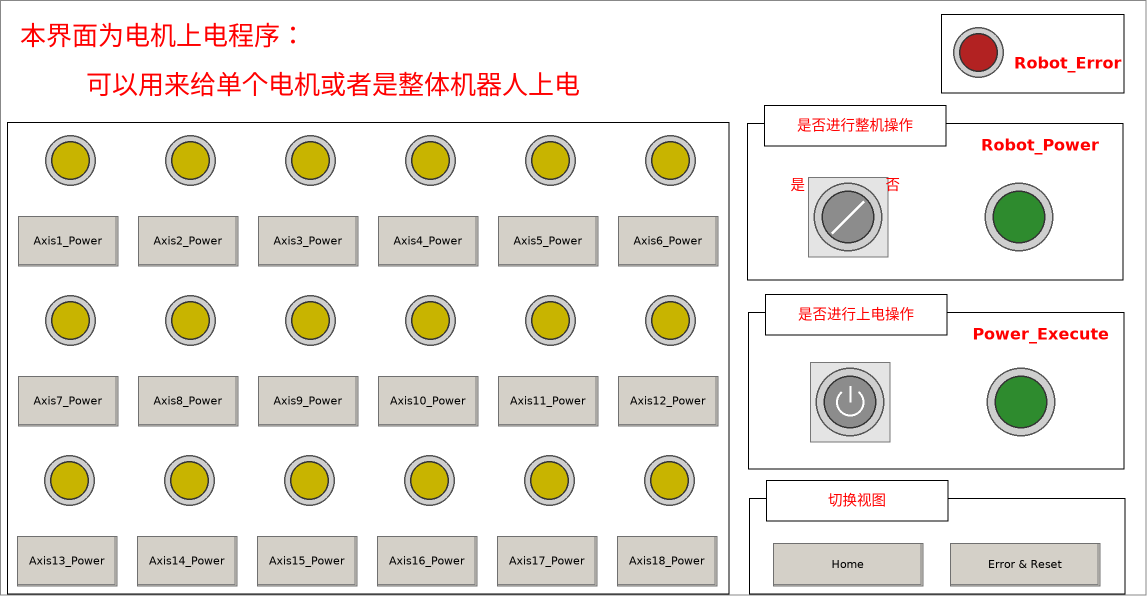
VISUALIZATION Visu_Power  // 1147x596
    Label (987,37 154x32), "Robot_Error"
    Rectangle (7,122 722x472)
    Lamp1 (40,131 61x59), variable: MAIN.Power_Status[1], style: Lamp-Lamp1-Yellow
    Lamp1 (160,131 61x59), variable: MAIN.Power_Status[2], style: Lamp-Lamp1-Yellow
    Lamp1 (280,131 61x59), variable: MAIN.Power_Status[3], style: Lamp-Lamp1-Yellow
    Lamp1 (400,131 61x59), variable: MAIN.Power_Status[4], style: Lamp-Lamp1-Yellow
    Lamp1 (520,131 61x59), variable: MAIN.Power_Status[5], style: Lamp-Lamp1-Yellow
    Lamp1 (640,131 61x59), variable: MAIN.Power_Status[6], style: Lamp-Lamp1-Yellow
    Button (18,216 100x50), "Axis1_Power"
        toggle MAIN.Axis_Power[1]
    Button (138,216 100x50), "Axis2_Power"
        toggle MAIN.Axis_Power[2]
    Button (258,216 100x50), "Axis3_Power"
        toggle MAIN.Axis_Power[3]
    Button (378,216 100x50), "Axis4_Power"
        toggle MAIN.Axis_Power[4]
    Button (498,216 100x50), "Axis5_Power"
        toggle MAIN.Axis_Power[5]
    Button (618,216 100x50), "Axis6_Power"
        toggle MAIN.Axis_Power[6]
    Lamp1 (40,291 61x59), variable: MAIN.Power_Status[7], style: Lamp-Lamp1-Yellow
    Lamp1 (160,291 61x59), variable: MAIN.Power_Status[8], style: Lamp-Lamp1-Yellow
    Lamp1 (280,291 61x59), variable: MAIN.Power_Status[9], style: Lamp-Lamp1-Yellow
    Lamp1 (400,291 61x59), variable: MAIN.Power_Status[10], style: Lamp-Lamp1-Yellow
    Lamp1 (520,291 61x59), variable: MAIN.Power_Status[11], style: Lamp-Lamp1-Yellow
    Lamp1 (640,291 61x59), variable: MAIN.Power_Status[12], style: Lamp-Lamp1-Yellow
    Button (18,376 100x50), "Axis7_Power"
        toggle MAIN.Axis_Power[7]
    Button (138,376 100x50), "Axis8_Power"
        toggle MAIN.Axis_Power[8]
    Button (258,376 100x50), "Axis9_Power"
        toggle MAIN.Axis_Power[9]
    Button (378,376 100x50), "Axis10_Power"
        toggle MAIN.Axis_Power[10]
    Button (498,376 100x50), "Axis11_Power"
        toggle MAIN.Axis_Power[11]
    Button (618,376 100x50), "Axis12_Power"
        toggle MAIN.Axis_Power[12]
    Lamp1 (39,451 61x59), variable: MAIN.Power_Status[13], style: Lamp-Lamp1-Yellow
    Lamp1 (159,451 61x59), variable: MAIN.Power_Status[14], style: Lamp-Lamp1-Yellow
    Lamp1 (279,451 61x59), variable: MAIN.Power_Status[15], style: Lamp-Lamp1-Yellow
    Lamp1 (399,451 61x59), variable: MAIN.Power_Status[16], style: Lamp-Lamp1-Yellow
    Lamp1 (519,451 61x59), variable: MAIN.Power_Status[17], style: Lamp-Lamp1-Yellow
    Lamp1 (639,451 61x59), variable: MAIN.Power_Status[18], style: Lamp-Lamp1-Yellow
    Button (17,536 100x50), "Axis13_Power"
        toggle MAIN.Axis_Power[13]
    Button (137,536 100x50), "Axis14_Power"
        toggle MAIN.Axis_Power[14]
    Button (257,536 100x50), "Axis15_Power"
        toggle MAIN.Axis_Power[15]
    Button (377,536 100x50), "Axis16_Power"
        toggle MAIN.Axis_Power[16]
    Button (497,536 100x50), "Axis17_Power"
        toggle MAIN.Axis_Power[17]
    Button (617,536 100x50), "Axis18_Power"
        toggle MAIN.Axis_Power[18]
    Rectangle (748,312 376x157)
    Label (964,318 154x32), "Power_Execute"
    Rectangle (765,294 182x41), "是否进行上电操作"
    Lamp1 (981,362 80x80), variable: MAIN.Power_Execute, style: Lamp-Lamp1-Green
    Rectangle (749,498 376x96)
    Rectangle (766,480 182x41), "切换视图"
    Button (773,543 150x43), "Home"
        OnMouseClick: change screen: Visu_Home
    PowerSwitch (810,362 80x80), variable: MAIN.Power_Execute, behaviour: TOGGLE, style: Switch-PowerSwitch-Gray
    Rectangle (941,14 183x79)
    Lamp1 (948,23 61x59), variable: MAIN.Robot_Error, style: Lamp-Lamp1-Red
    Label (17,15 365x42), "本界面为电机上电程序："
    Label (83,64 639x42), "可以用来给单个电机或者是整体机器人上电"
    Button (950,543 150x43), "Error & Reset"
        OnMouseClick: change screen: Visu_Reset
    Rectangle (747,123 376x157)
    Label (963,129 154x32), "Robot_Power"
    Rectangle (764,105 182x41), "是否进行整机操作"
    Lamp1 (979,177 80x80), variable: MAIN.Robot_Power, style: Lamp-Lamp1-Green
    RotarySwitch (808,177 80x80), variable: MAIN.Robot_Power, behaviour: TOGGLE, style: Switch-RotarySwitch-Gray
    Label (863,170 60x30), "否"
    Label (768,170 60x30), "是"
    Label (991,47 154x32), "Robot_Error"
END_VISUALIZATION

(* stored: Version 1.1.0.1, ProductVersion 3.1.4020.12
   Visu Visu_Power: Id {58811ec6-071b-47ae-a16b-4b1b3a9b4cdb} *)
